// TIA Portal V16 export
// export: Created 2025-08-01T13:37:56.4100405Z, ExportSetting WithDefaults, DisplayName Totally Integrated Automation Portal, DisplayVersion V16, DisplayName TIA Portal Version Control Interface, DisplayVersion V16, DisplayName TIA Portal Openness, DisplayVersion V16, DisplayName STEP 7 Professional, DisplayVersion V16, DisplayName STEP 7 Safety, DisplayVersion V16, DisplayName WinCC Advanced, DisplayVersion V16
FUNCTION "7 - Clean" : Void   // FC4, LAD
TITLE = Cleaning Program
VERSION : 0.1
// stored: AutoNumber true, IsIECCheckEnabled false, UDAEnableTagReadback false
   VAR_TEMP
      BlowOff_Active : Bool;
   END_VAR
   VAR_TEMP   // added for the SCL form of the ladder/FBD networks
      _w1 : Bool;
   END_VAR
BEGIN

REGION Network 1: Button Pressed Show Message
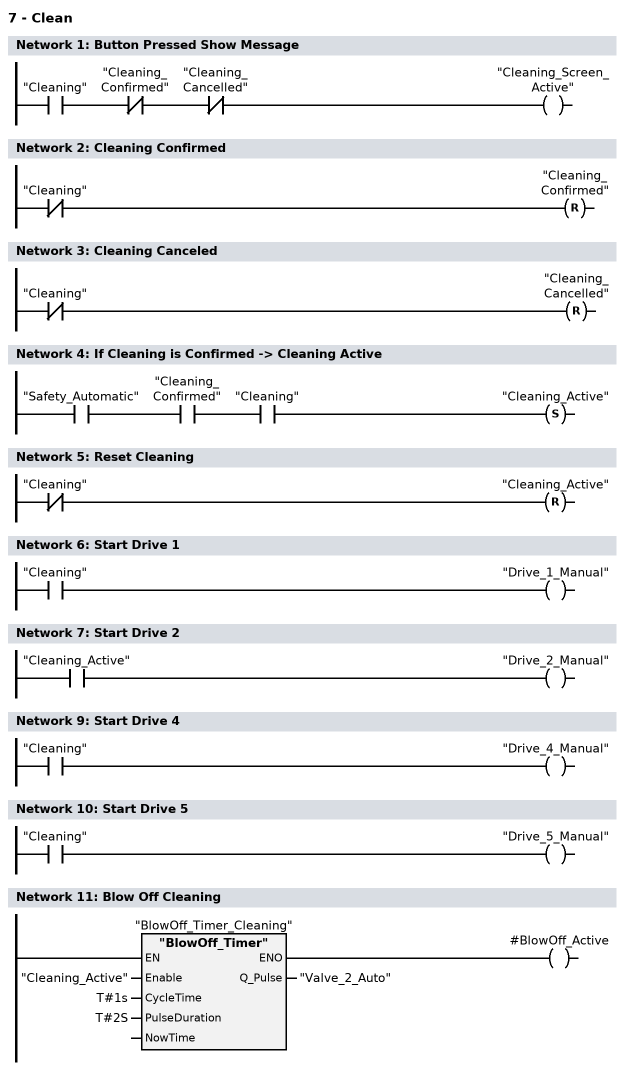
   RUNG wire#powerrail
      Contact( "Cleaning" )
      I_Contact( "Cleaning_Confirmed" )
      I_Contact( "Cleaning_Cancelled" )
      Coil( "Cleaning_Screen_Active" )
   END_RUNG
   // the same network as SCL:
   "Cleaning_Screen_Active" := "Cleaning" AND NOT "Cleaning_Confirmed" AND NOT "Cleaning_Cancelled";
END_REGION

REGION Network 2: Cleaning Confirmed
   RUNG wire#powerrail
      I_Contact( "Cleaning" )
      R_Coil( "Cleaning_Confirmed" )
   END_RUNG
   // the same network as SCL:
   IF NOT "Cleaning" THEN "Cleaning_Confirmed" := FALSE; END_IF;
END_REGION

REGION Network 3: Cleaning Canceled
   RUNG wire#powerrail
      I_Contact( "Cleaning" )
      R_Coil( "Cleaning_Cancelled" )
   END_RUNG
   // the same network as SCL:
   IF NOT "Cleaning" THEN "Cleaning_Cancelled" := FALSE; END_IF;
END_REGION

REGION Network 4: If Cleaning is Confirmed -> Cleaning Active
   RUNG wire#powerrail
      Contact( "Safety_Automatic" )
      Contact( "Cleaning_Confirmed" )
      Contact( "Cleaning" )
      S_Coil( "Cleaning_Active" )
   END_RUNG
   // the same network as SCL:
   IF "Safety_Automatic" AND "Cleaning_Confirmed" AND "Cleaning" THEN "Cleaning_Active" := TRUE; END_IF;
END_REGION

REGION Network 5: Reset Cleaning
   RUNG wire#powerrail
      I_Contact( "Cleaning" )
      R_Coil( "Cleaning_Active" )
   END_RUNG
   // the same network as SCL:
   IF NOT "Cleaning" THEN "Cleaning_Active" := FALSE; END_IF;
END_REGION

REGION Network 6: Start Drive 1
   RUNG wire#powerrail
      Contact( "Cleaning" )
      Coil( "Drive_1_Manual" )
   END_RUNG
   // the same network as SCL:
   "Drive_1_Manual" := "Cleaning";
END_REGION

REGION Network 7: Start Drive 2
   RUNG wire#powerrail
      Contact( "Cleaning_Active" )
      Coil( "Drive_2_Manual" )
   END_RUNG
   // the same network as SCL:
   "Drive_2_Manual" := "Cleaning_Active";
END_REGION

REGION Network 8: Start Drive 3
END_REGION

REGION Network 9: Start Drive 4
   RUNG wire#powerrail
      Contact( "Cleaning" )
      Coil( "Drive_4_Manual" )
   END_RUNG
   // the same network as SCL:
   "Drive_4_Manual" := "Cleaning";
END_REGION

REGION Network 10: Start Drive 5
   RUNG wire#powerrail
      Contact( "Cleaning" )
      Coil( "Drive_5_Manual" )
   END_RUNG
   // the same network as SCL:
   "Drive_5_Manual" := "Cleaning";
END_REGION

REGION Network 11: Blow Off Cleaning
   RUNG wire#powerrail
      "BlowOff_Timer_Cleaning"(Enable := "Cleaning_Active", CycleTime := T#1s, PulseDuration := T#2S, Q_Pulse => "Valve_2_Auto", NowTime :=)
      Coil( #BlowOff_Active )
   END_RUNG
   // the same network as SCL:
   "BlowOff_Timer_Cleaning"(Enable := "Cleaning_Active",   // "BlowOff_Timer"
                           CycleTime := T#1s,
                           PulseDuration := T#2S,
                           Q_Pulse => "Valve_2_Auto",
                           ENO => #_w1);
   #BlowOff_Active := #_w1;
END_REGION
END_FUNCTION
